INTERFACE ITF_EM_Transport_TurningDevice_StampUnit

END_INTERFACE

(* stored: Version 1.1.0.1, ProductVersion 3.1.4024.12
   Itf ITF_EM_Transport_TurningDevice_StampUnit: Id {84c8723a-7154-4707-8580-92c67d482257} *)
